RoboDK station: Proyecto.rdk

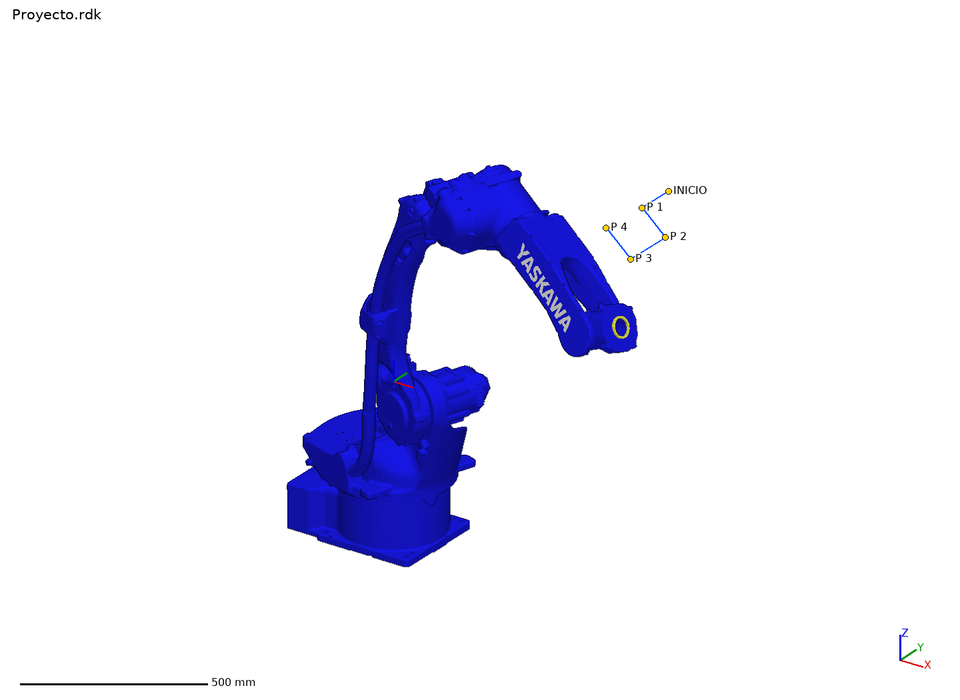
[picture v0: the station drawn from its stored meshes, robots at their saved joint values, targets as dots, program paths as lines]
Station Proyecto (saved by RoboDK 5.7.5). Poses are relative to the parent item; angles as X-Y-Z fixed-axis rotations.
  - frame Yaskawa AR1440 Base at (0, 0, 450) mm
    - robot Yaskawa AR1440: 6 axes
        modified DH rows (alpha deg, a mm, theta deg, d mm): 0, 0, 0, 450; -90, 155, -90, 0; 0, 614, 0, 0; -90, 200, 0, 640; 90, 0, 0, 0; -90, 0, 180, 100
        base shift (0, 0, -450) mm
        joint limits [-170, -90, -85, -150, -135, -210] to [170, 155, 140, 150, 90, 210]; home [0, 0, 0, 0, 0, 0]; saved at [-19.174, 9.182, 16.327, -18.342, -51.582, 24.578]
    - target INICIO (Cartesian target) at (895, 0, 814) mm, rotated rx 180 ry -48.65 rz 0 deg; joints [0, 4.704, 10.921, 0, -47.565, 0] of Yaskawa AR1440
    - target P 1 (Cartesian target) at (895, -123.18, 814) mm, rotated rx -180 ry -48.65 rz 0 deg; joints [-8.544, 5.601, 11.899, -8.593, -48.284, 11.41] of Yaskawa AR1440
    - target P 2 (Cartesian target) at (970.56, -123.18, 747.5) mm, rotated rx -180 ry -48.65 rz 0 deg; joints [-7.832, 10.52, 11.407, -8.655, -42.828, 11.563] of Yaskawa AR1440
    - target P 3 (Cartesian target) at (970.56, -283.48, 747.5) mm, rotated rx -180 ry -48.65 rz 0 deg; joints [-17.566, 14.167, 15.808, -18.406, -45.853, 24.862] of Yaskawa AR1440
    - target P 4 (Cartesian target) at (890.32, -283.48, 818.12) mm, rotated rx -180 ry -48.65 rz 0 deg; joints [-19.174, 9.182, 16.327, -18.342, -51.582, 24.578] of Yaskawa AR1440
  - program Prog1 (6 instructions, listed below)
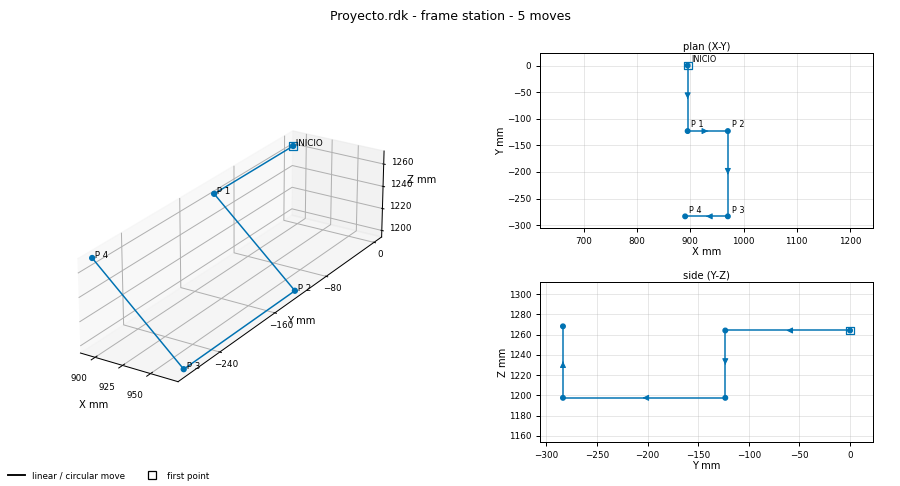
[picture p0: tool path of Proyecto.rdk in frame station, 5 of 5 moves have a stored position in this frame; points joined in program order, loops and branches not executed]

--- program Prog1 (robot Yaskawa AR1440) ---
  Est. Ref.: Yaskawa AR1440 Base
  MoveJ (INICIO)
  MoveL (P 1)
  MoveL (P 2)
  MoveL (P 3)
  MoveL (P 4)
